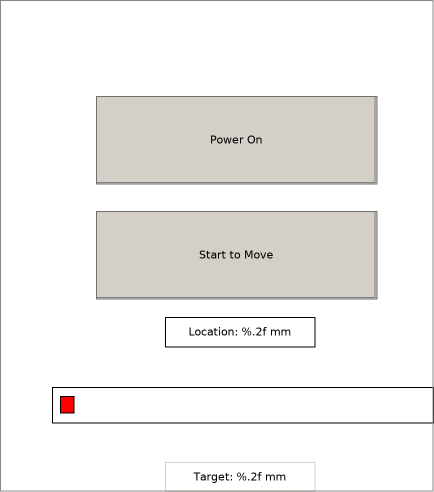
VISUALIZATION HomeScreen  // 434x492
    Button (96,96 281x88), "Power On"
        toggle MAIN.bEnable
    Button (96,211 281x88), "Start to Move"
        toggle MAIN.bMoveStart
    Rectangle (165,317 150x30), "Location: %.2f mm", text variable: MAIN.fLocation
    Textfield (165,462 150x30), "Target: %.2f mm", text variable: MAIN.fTargetLocation
        OnMouseClick: write the text variable via VisuDialogs.Numpad
    Rectangle (52,387 382x36)
    Rectangle (60,396 14x17)
        p3560616238: MAIN.fLocation
END_VISUALIZATION

(* stored: Version 1.1.0.1
   Visu HomeScreen: Id {87a5b859-8378-4315-937d-c451e68caa1e} *)
